(* Logix 5000 project; controller PBS_Perfusion vendor 1 type 14 code 217 rev 32.14; software revision 32.03; part 20 of 27 *)
(* tags used below, declared in another part *)
   Inp_PermOK : BOOL;   // 1=Permissives OK, Valve can energize
   Inp_NBPermOK : BOOL;   // 1=Non-Bypassable Permissives OK, valve can energize
   Inp_IOFault : BOOL;   // Input Communication Status 0=OK, 1=fail
   Inp_Sim : BOOL;   // 1=Simulate working valve; 0=Open/Close/ Monitor actual valve
   Inp_OvrdCmd : DINT;   // Override Mode Command: 0=None, 1=Close, 2=Open
   Cfg_FailOpen : BOOL;   // 1=Fail Open (energize to close), 0=Fail Closed (energize to open)
   Cfg_HasOpenLS : BOOL;   // 1=Valve provides an Open Limit Switch signal
   Cfg_HasClosedLS : BOOL;   // 1=Valve provides a Closed Limit Switch signal
   Cfg_UseOpenLS : BOOL;   // 1=Valve Open LS should be used for failure checking
   Cfg_UseClosedLS : BOOL;   // 1=Valve Closed LS should be used for failure checking
   Cfg_OCmdResets : BOOL;   // 1=New valve OCmd resets shed latches and cleared alarms, 0=OCmdReset req'd.
   PSet_Owner : DINT;   // Program Owner Request ID (non-zero) or Release (zero)
   PCmd_Open : BOOL;   // Program Command to Open Valve
   PCmd_Close : BOOL;   // Program Command to Close Valve
   PCmd_Reset : BOOL;   // Program Command to ResetShed Latches and Cleared Alarms
   XCmd_Open : BOOL;   // External Command to Open Valve
   XCmd_Close : BOOL;   // External Command to Close Valve
   XCmd_Reset : BOOL;   // Ext Cmd to clear shed latches and cleared alarms
   Out : BOOL;   // 1=Energize Valve Solenoid
   Out_Horn : BOOL;   // 1=Sound audible prior to commanded motor start
   SrcQ_IO : DINT;   // Source and Quality of primary I/O (enumeration)
   SrcQ : DINT;   // Source and Quality of primary Val/Sts (enumeration)
   Val_Cmd : DINT;   // Device Command 0=None, 1=Close, 2=Open
   Val_Fdbk : DINT;   // Device Feedback 0=Moving, 1=Closed, 2=Opened, 3=Limit Switch Failure
   Val_Sts : DINT;   // Device Confirmed Sts 0=? 1=Closed 2=Open 5=Closing, 6=Opening
   Val_Fault : DINT;   // Device Fault Status 0=None, 16=Transit Stall, 17 = Full Stall, 32=I/O Fault, 34=Config Error
   Val_NotifyAll : DINT;   // Highest Alarm prio and ack status this object + channel (enum)
   Val_UnackAlmC : DINT;   // Count of Unacknowledged Alarms
   Val_Owner : DINT;   // Current Object Owner ID (0=not owned)
   Sts_Closed : BOOL;   // 1=Valve requested to Close and is confirmed Closed
   Sts_Opening : BOOL;   // 1=Valve requested to open and awaiting open feedback
   Sts_Opened : BOOL;   // 1=Valve requested to open and is confirmed Opened
   Sts_Closing : BOOL;   // 1=Valve requested to Close and awaiting Closed feedback
   Sts_Horn : BOOL;   // 1=Valve Horn Active
   Sts_BypActive : BOOL;   // 1=Bypassing Active (Bypassed or Maintenance)
   Sts_NotRdy : BOOL;   // 1=Device Not Ready, see detail bits for reason
   Nrdy_CfgErr : BOOL;   // 1=Device Not Ready: Configuration Error
   Nrdy_Fail : BOOL;   // 1=Device Not Ready: Device Failure (Shed Requires Reset)
   Nrdy_IOFault : BOOL;   // 1=Device Not Ready: I/O Fault (Shed Requires Reset)
   Sts_AlmInh : BOOL;   // 1=An Alarm is Shelved, Disabled or Suppressed, display icon
   Sts_Err : BOOL;   // 1=Error in Config: see detail bits for reason
   Err_Alarm : BOOL;   // 1=Error in Config: Alarm Min On Time, Shelf Time, Severity
   Sts_Hand : ALIAS FOR CmdSrc.Sts_Hand;
   Sts_OoS : ALIAS FOR CmdSrc.Sts_OoS;
   Sts_Maint : ALIAS FOR CmdSrc.Sts_Maint;
   Sts_Oper : ALIAS FOR CmdSrc.Sts_Oper;
   Sts_RdyReset : ALIAS FOR ORdy_Reset;   // 1=A latched alarm or shed condition is ready to be reset
   Sts_RdyAck : BOOL;   // 1=An alarm is ready to be acknowledged
   Sts_FullStall : ALIAS FOR FullStall.Inp;   // 1=Valve Full Stall (failed to move at all)
   Sts_TransitStall : ALIAS FOR TransitStall.Inp;   // 1=Valve Transit Stall (did not reach target position)
   Sts_IOFault : ALIAS FOR IOFault.Inp;   // I/O Comm Fault Status (0=OK, 1=Bad)
   P_ValveSO : BOOL;   // Unique Parameter Name for auto - discovery
   CmdSrc : P_CmdSrc;   // Valve Mode Selection
   IOFault : P_Alarm;   // I/O Fault Alarm
   IntlkTrip : P_Alarm;   // Interlock Trip Alarm
   TransitStall : P_Alarm;   // Valve Transit Stall (moved but did not reach target) Alarm
   FullStall : P_Alarm;   // Valve Full Stall (did not move) Alarm
   Wrk_Open : BOOL;   // 1=Requested to OPEN Valve, 0=Requested to CLOSE Valve
   Wrk_SimOpenT : TIMER;   // Simulation Delay until Opened
   Wrk_SimCloseT : TIMER;   // Simulation Delay until Closed
   Wrk_OpenFdbk : BOOL;   // 1=LS Feedback shows valve confirmed open
   Wrk_Notify : DINT;   // Buffer for building Val_Notify
   Wrk_ClosedFdbk : BOOL;   // 1=LS Feedback shows valve confirmed closed
   Wrk_TransitStallT : TIMER;   // Timer for Transit Stall Check
   Wrk_FullStallT : TIMER;   // Timer for Full Stall Check
   Wrk_Cmd : DINT;   // Buffer for building Val_Cmd
   Wrk_Sts : DINT;   // Buffer for building Val_Sts
   Wrk_Fault : DINT;   // Buffer for building Val_Fault
   Wrk_SimOpenLS : BOOL;   // Simulated valve Open Limit Switch
   Wrk_SimClosedLS : BOOL;   // Simulated valve Closed Limit Switch
   Wrk_SrcQ : DINT;   // Register for building Source / Quality enumeration
   Val_Notify : DINT;   // Current Alarm Level and Acknowledgement (enumeration)
   Wrk_NotRdy : BOOL;   // Device Not Ready conditions excluding shed latches
   Wrk_NoLongerSim : BOOL;   // Switched from Simulated to Real Valve this scan
   OCmd_Close : BOOL;   // Operator Command to Close Valve
   OCmd_Open : BOOL;   // Operator Command to Open Valve
   ORdy_ResetAckAll : BOOL;   // 1=Ready for OCmd_ResetAckAll (enables HMI button)
   ORdy_Reset : BOOL;   // 1=Ready for OCmd_Reset (enables HMI button)
   MRdy_Check : BOOL;   // 1=Ready for MCmd_Check (enables HMI button)
   MRdy_Bypass : BOOL;   // 1=Ready for MCmd_Bypass (enables HMI button)
   ORdy_Close : BOOL;   // 1=Ready for OCmd_Close (enables HMI button)
   ORdy_Open : BOOL;   // 1=Ready for OCmd_Open (enables HMI button)
   MCmd_Check : BOOL;   // Maintenance Command to Check (not bypass) all Interlocks and Permissives
   MCmd_Bypass : BOOL;   // Maintenance Command to Bypass all Bypassable Interlocks and Permissives
   OCmd_ResetAckAll : BOOL;   // Oper Cmd to reset shed latches and cleared alarms, plus Acknowledge alarms
   OCmd_Reset : BOOL;   // Oper Cmd to clear shed latches and cleared alarms
   Wrk_UnackAlmC : DINT;   // Buffer for building Val_UnackAlmC
   Wrk_CloseCmdRcvd : BOOL;   // 1=Received a Close command this scan
   Wrk_OpenCmdRcvd : BOOL;   // 1=Received an Open command this scan
   Wrk_StartHornT : TIMER;   // Timer for audible alert on start
   Wrk_StartHorn : BOOL;   // 1=Sound audible prior to commanded motor start
   ONS : DINT[3];
(* P_ValveSO, continued *)

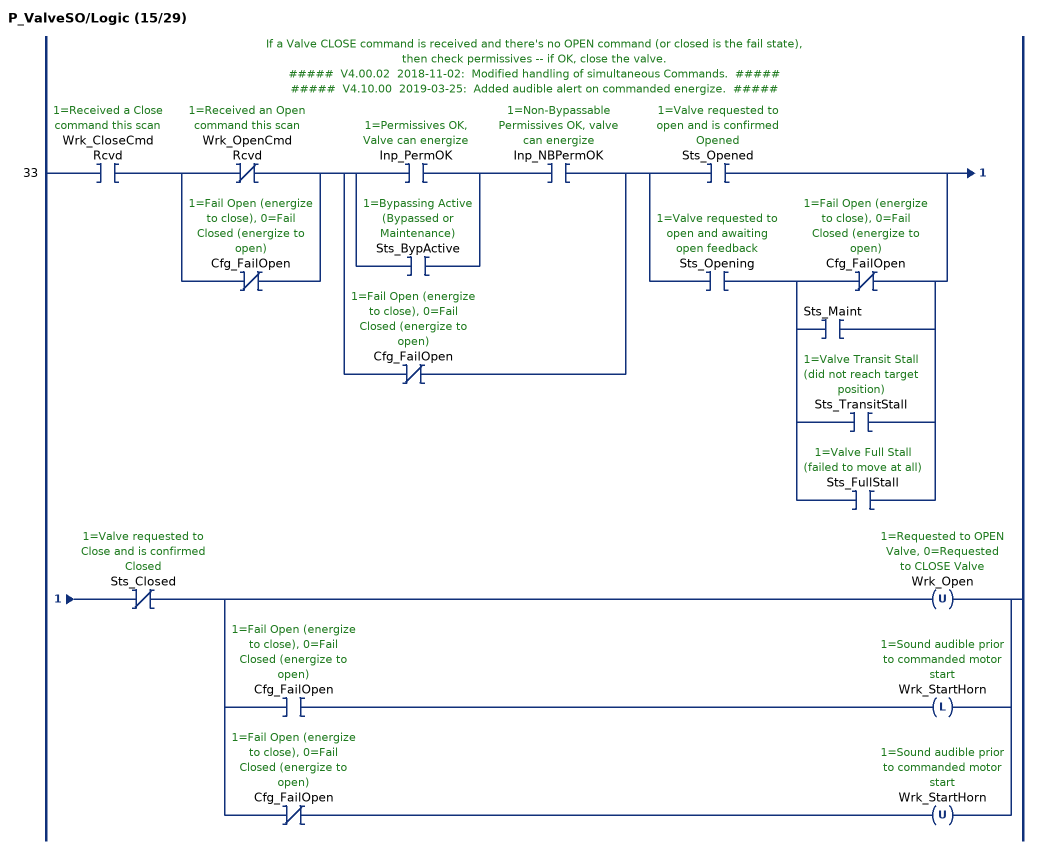
   [picture p443: P_ValveSO/Logic rungs 33-33]
   // If a Valve CLOSE command is received and there's no OPEN command (or closed is the fail state),
   // then check permissives -- if OK, close the valve.
   // #####  V4.00.02  2018-11-02:  Modified handling of simultaneous Commands.  #####
   // #####  V4.10.00  2019-03-25:  Added audible alert on commanded energize.  #####
   33: XIC(Wrk_CloseCmdRcvd)[XIO(Wrk_OpenCmdRcvd) ,XIO(Cfg_FailOpen) ][[XIC(Inp_PermOK) ,XIC(Sts_BypActive) ] XIC(Inp_NBPermOK) ,XIO(Cfg_FailOpen) ][XIC(Sts_Opened) ,XIC(Sts_Opening) [XIO(Cfg_FailOpen) ,XIC(Sts_Maint) ,XIC(Sts_TransitStall) ,XIC(Sts_FullStall) ] ]XIO(Sts_Closed)[OTU(Wrk_Open) ,XIC(Cfg_FailOpen) OTL(Wrk_StartHorn) ,XIO(Cfg_FailOpen) OTU(Wrk_StartHorn) ];
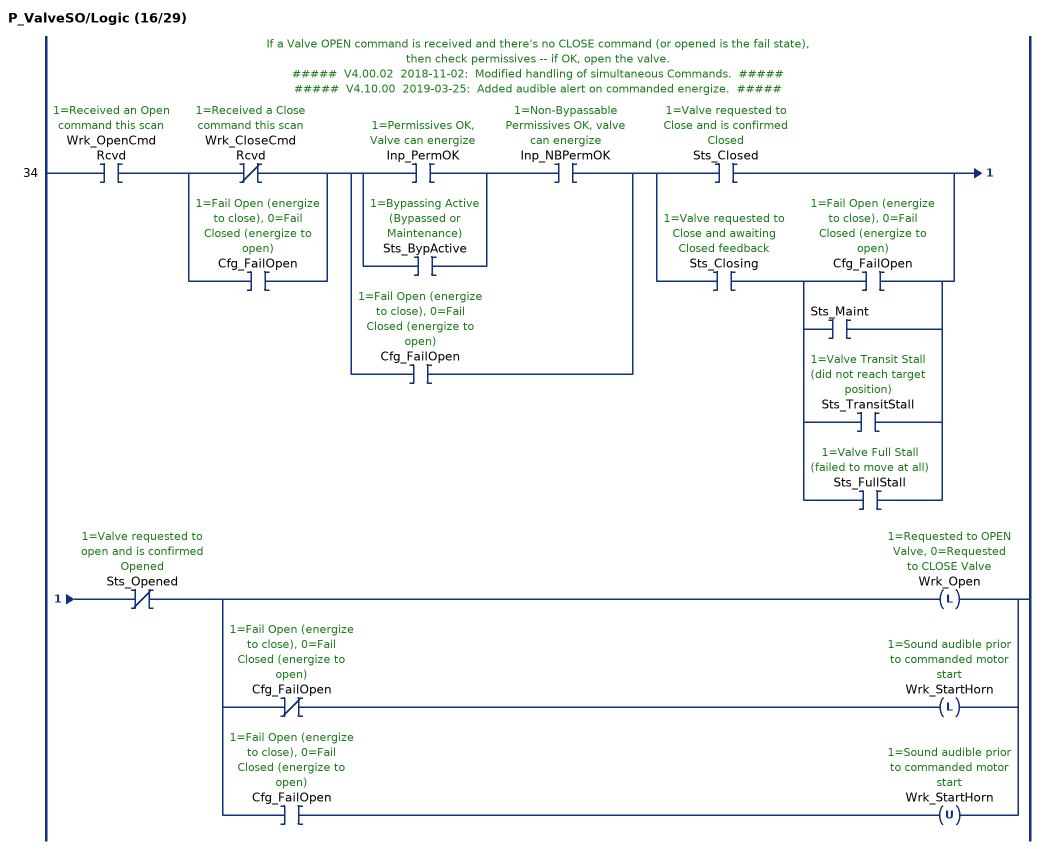
   // If a Valve OPEN command is received and there's no CLOSE command (or opened is the fail state),
   // then check permissives -- if OK, open the valve.
   // #####  V4.00.02  2018-11-02:  Modified handling of simultaneous Commands.  #####
   // #####  V4.10.00  2019-03-25:  Added audible alert on commanded energize.  #####
   34: XIC(Wrk_OpenCmdRcvd)[XIO(Wrk_CloseCmdRcvd) ,XIC(Cfg_FailOpen) ][[XIC(Inp_PermOK) ,XIC(Sts_BypActive) ] XIC(Inp_NBPermOK) ,XIC(Cfg_FailOpen) ][XIC(Sts_Closed) ,XIC(Sts_Closing) [XIC(Cfg_FailOpen) ,XIC(Sts_Maint) ,XIC(Sts_TransitStall) ,XIC(Sts_FullStall) ] ]XIO(Sts_Opened)[OTL(Wrk_Open) ,XIO(Cfg_FailOpen) OTL(Wrk_StartHorn) ,XIC(Cfg_FailOpen) OTU(Wrk_StartHorn) ];
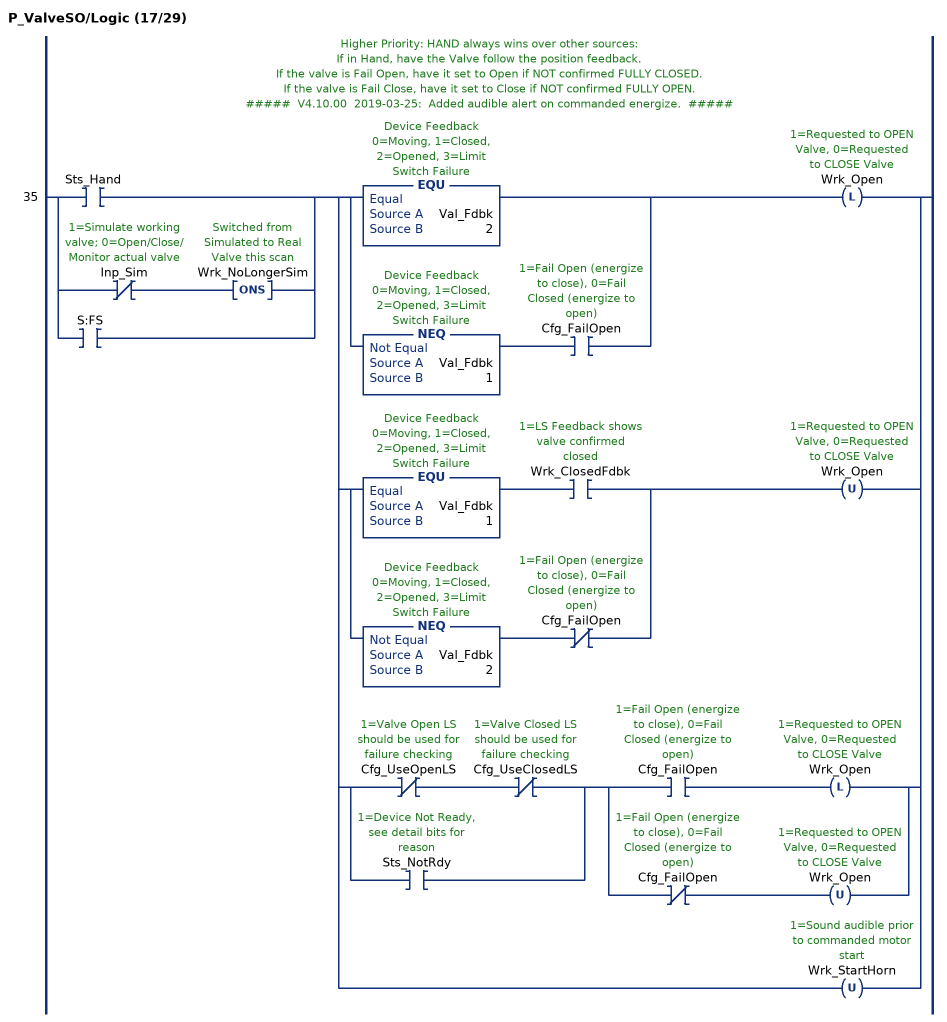
   // Higher Priority: HAND always wins over other sources:
   // If in Hand, have the Valve follow the position feedback.
   // If the valve is Fail Open, have it set to Open if NOT confirmed FULLY CLOSED.
   // If the valve is Fail Close, have it set to Close if NOT confirmed FULLY OPEN.
   // #####  V4.10.00  2019-03-25:  Added audible alert on commanded energize.  #####
   35: [XIC(Sts_Hand) ,XIO(Inp_Sim) ONS(Wrk_NoLongerSim) ,XIC(S:FS) ][[EQU(Val_Fdbk,2) ,NEQ(Val_Fdbk,1) XIC(Cfg_FailOpen) ] OTL(Wrk_Open) ,[EQU(Val_Fdbk,1) XIC(Wrk_ClosedFdbk) ,NEQ(Val_Fdbk,2) XIO(Cfg_FailOpen) ] OTU(Wrk_Open) ,[XIO(Cfg_UseOpenLS) XIO(Cfg_UseClosedLS) ,XIC(Sts_NotRdy) ] [XIC(Cfg_FailOpen) OTL(Wrk_Open) ,XIO(Cfg_FailOpen) OTU(Wrk_Open) ] ,OTU(Wrk_StartHorn) ];
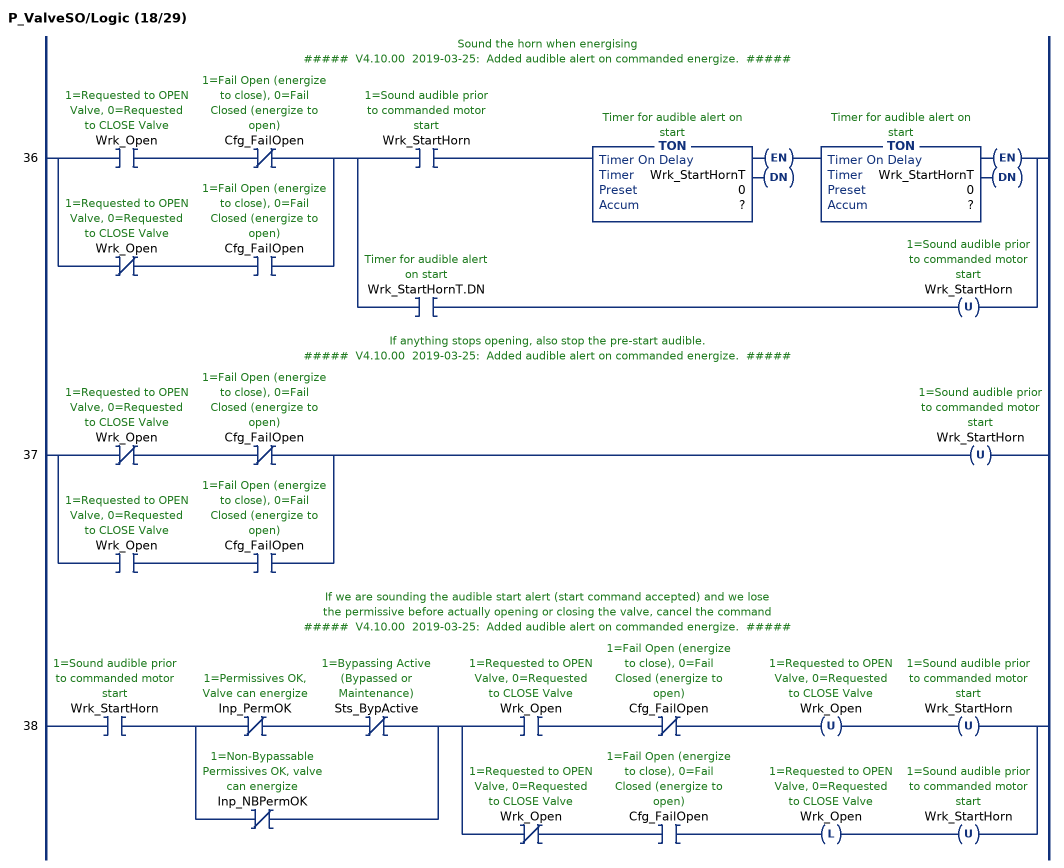
   // Sound the horn when energising
   // #####  V4.10.00  2019-03-25:  Added audible alert on commanded energize.  #####
   36: [XIC(Wrk_Open) XIO(Cfg_FailOpen) ,XIO(Wrk_Open) XIC(Cfg_FailOpen) ][XIC(Wrk_StartHorn) TON(Wrk_StartHornT,?,?) TON(Wrk_StartHornT,?,?) ,XIC(Wrk_StartHornT.DN) OTU(Wrk_StartHorn) ];
   // If anything stops opening, also stop the pre-start audible.
   // #####  V4.10.00  2019-03-25:  Added audible alert on commanded energize.  #####
   37: [XIO(Wrk_Open) XIO(Cfg_FailOpen) ,XIC(Wrk_Open) XIC(Cfg_FailOpen) ]OTU(Wrk_StartHorn);
   // If we are sounding the audible start alert (start command accepted) and we lose
   // the permissive before actually opening or closing the valve, cancel the command
   // #####  V4.10.00  2019-03-25:  Added audible alert on commanded energize.  #####
   38: XIC(Wrk_StartHorn)[XIO(Inp_PermOK) XIO(Sts_BypActive) ,XIO(Inp_NBPermOK) ][XIC(Wrk_Open) XIO(Cfg_FailOpen) OTU(Wrk_Open) OTU(Wrk_StartHorn) ,XIO(Wrk_Open) XIC(Cfg_FailOpen) OTL(Wrk_Open) OTU(Wrk_StartHorn) ];
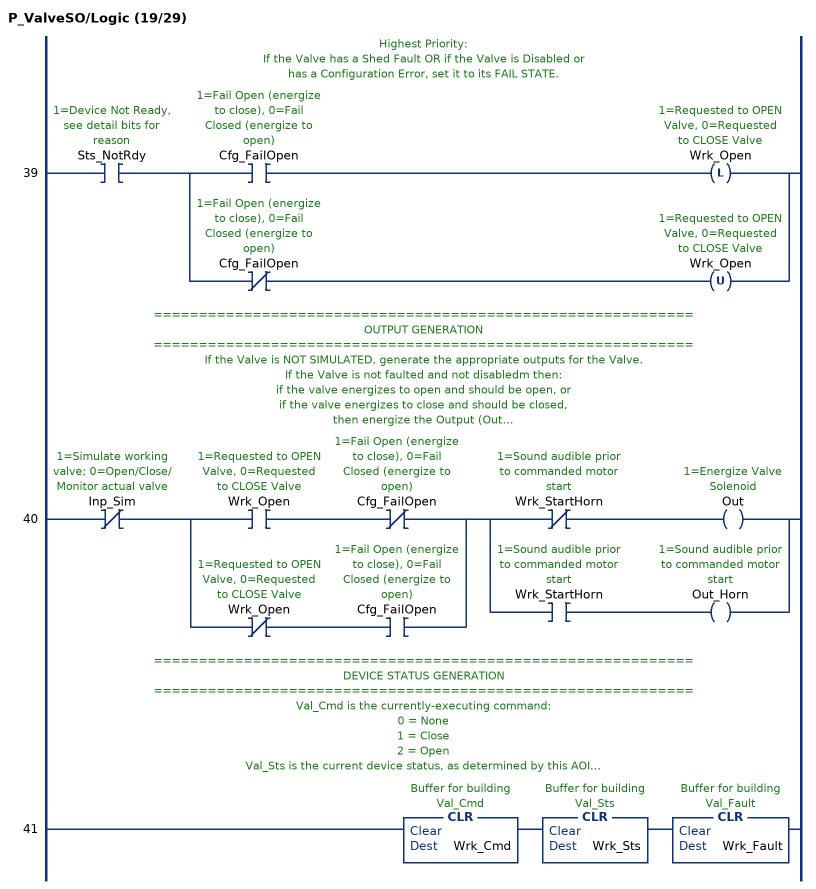
   // Highest Priority:
   // If the Valve has a Shed Fault OR if the Valve is Disabled or
   // has a Configuration Error, set it to its FAIL STATE.
   39: XIC(Sts_NotRdy)[XIC(Cfg_FailOpen) OTL(Wrk_Open) ,XIO(Cfg_FailOpen) OTU(Wrk_Open) ];
   // ============================================================
   // OUTPUT GENERATION
   // ============================================================
   // If the Valve is NOT SIMULATED, generate the appropriate outputs for the Valve.
   // If the Valve is not faulted and not disabledm then:
   // if the valve energizes to open and should be open, or
   // if the valve energizes to close and should be closed,
   // then energize the Output (Out)
   // #####  V4.10.00  2019-03-25:  Added audible alert on commanded energize.  #####
   40: XIO(Inp_Sim)[XIC(Wrk_Open) XIO(Cfg_FailOpen) ,XIO(Wrk_Open) XIC(Cfg_FailOpen) ][XIO(Wrk_StartHorn) OTE(Out) ,XIC(Wrk_StartHorn) OTE(Out_Horn) ];
   // ============================================================
   // DEVICE STATUS GENERATION
   // ============================================================
   // Val_Cmd is the currently-executing command:
   // 0 = None
   // 1 = Close
   // 2 = Open
   // Val_Sts is the current device status, as determined by this AOI,
   // based on its knowledge of commands executed and feedback.
   // (This is the status that should be monitored by, for example, FT Historian.)
   // 0 = Powerup / Unknown
   // 1 = Closed
   // 2 = Opened
   // 5 = Closing
   // 6 = Opening
   // 10 = Horn
   // 33 = Out of Service
   // Val_Fault is the current device fault status, as determined by this AOI,
   // based on its knowledge of commands executed and feedback.
   // (This is the fault status that should be monitored by, for example, FT Historian.)
   // 0 = None
   // 16 = Full Stall
   // 17 = Transit Stall
   // 32 = I/O Fault (from Input)
   // 34 = Configuration Error
   // #####  V4.10.00  2019-03-25:  Added Horn Status.  #####
   41: CLR(Wrk_Cmd)CLR(Wrk_Sts)CLR(Wrk_Fault);
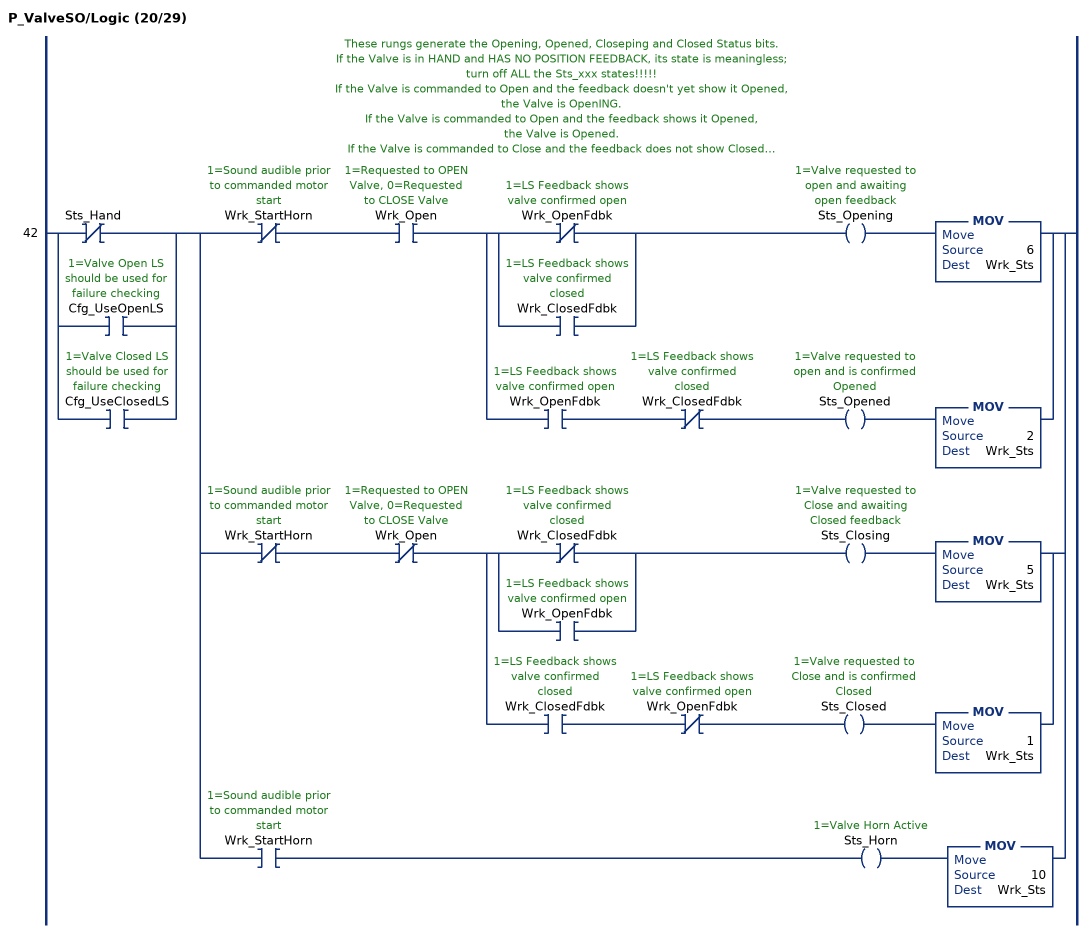
   // These rungs generate the Opening, Opened, Closeping and Closed Status bits.
   // If the Valve is in HAND and HAS NO POSITION FEEDBACK, its state is meaningless;
   // turn off ALL the Sts_xxx states!!!!!
   // If the Valve is commanded to Open and the feedback doesn't yet show it Opened,
   // the Valve is OpenING.
   // If the Valve is commanded to Open and the feedback shows it Opened,
   // the Valve is Opened.
   // If the Valve is commanded to Close and the feedback does not show Closed,
   // the Valve is CloseING.
   // If the Valve is commanded to Close and the feedback shows it has Closed,
   // the Valve is Closed.
   // If the audible alert is active, show the Status as HORN.
   // #####  V4.10.00  2019-03-25:  Added Horn Status.  #####
   42: [XIO(Sts_Hand) ,XIC(Cfg_UseOpenLS) ,XIC(Cfg_UseClosedLS) ][XIO(Wrk_StartHorn) XIC(Wrk_Open) [[XIO(Wrk_OpenFdbk) ,XIC(Wrk_ClosedFdbk) ] OTE(Sts_Opening) MOV(6,Wrk_Sts) ,XIC(Wrk_OpenFdbk) XIO(Wrk_ClosedFdbk) OTE(Sts_Opened) MOV(2,Wrk_Sts) ] ,XIO(Wrk_StartHorn) XIO(Wrk_Open) [[XIO(Wrk_ClosedFdbk) ,XIC(Wrk_OpenFdbk) ] OTE(Sts_Closing) MOV(5,Wrk_Sts) ,XIC(Wrk_ClosedFdbk) XIO(Wrk_OpenFdbk) OTE(Sts_Closed) MOV(1,Wrk_Sts) ] ,XIC(Wrk_StartHorn) OTE(Sts_Horn) MOV(10,Wrk_Sts) ];
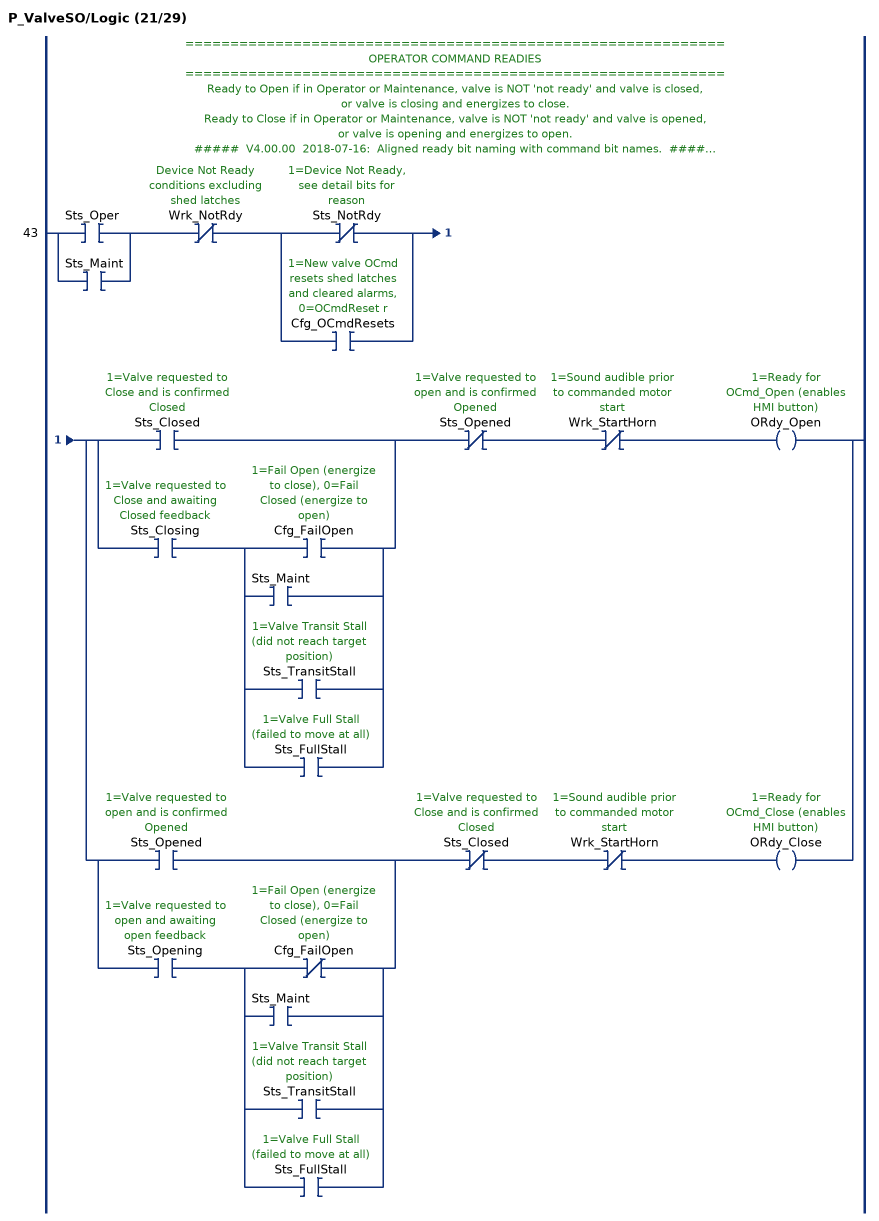
   // ============================================================
   // OPERATOR COMMAND READIES
   // ============================================================
   // Ready to Open if in Operator or Maintenance, valve is NOT 'not ready' and valve is closed,
   // or valve is closing and energizes to close.
   // Ready to Close if in Operator or Maintenance, valve is NOT 'not ready' and valve is opened,
   // or valve is opening and energizes to open.
   // #####  V4.00.00  2018-07-16:  Aligned ready bit naming with command bit names.  #####
   // #####  V4.10.00  2019-03-25:  Added audible alert on commanded energize.  #####
   43: [XIC(Sts_Oper) ,XIC(Sts_Maint) ]XIO(Wrk_NotRdy)[XIO(Sts_NotRdy) ,XIC(Cfg_OCmdResets) ][[XIC(Sts_Closed) ,XIC(Sts_Closing) [XIC(Cfg_FailOpen) ,XIC(Sts_Maint) ,XIC(Sts_TransitStall) ,XIC(Sts_FullStall) ] ] XIO(Sts_Opened) XIO(Wrk_StartHorn) OTE(ORdy_Open) ,[XIC(Sts_Opened) ,XIC(Sts_Opening) [XIO(Cfg_FailOpen) ,XIC(Sts_Maint) ,XIC(Sts_TransitStall) ,XIC(Sts_FullStall) ] ] XIO(Sts_Closed) XIO(Wrk_StartHorn) OTE(ORdy_Close) ];
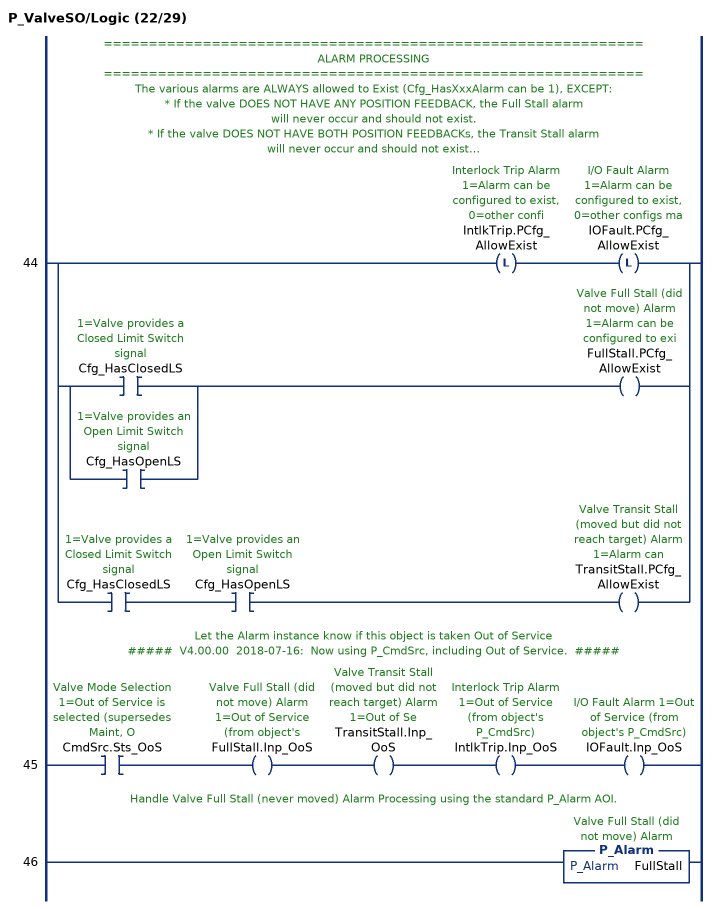
   // ============================================================
   // ALARM PROCESSING
   // ============================================================
   // The various alarms are ALWAYS allowed to Exist (Cfg_HasXxxAlarm can be 1), EXCEPT:
   // * If the valve DOES NOT HAVE ANY POSITION FEEDBACK, the Full Stall alarm
   // will never occur and should not exist.
   // * If the valve DOES NOT HAVE BOTH POSITION FEEDBACKs, the Transit Stall alarm
   // will never occur and should not exist.
   // (If feedback exists, the stall alarms must be allowed to exist.)
   // #####  V4.00.00  2018-07-16:  Deleted Cfg_PCmdClear; all Program Commands are now self-clearing.  #####
   44: [OTL(IntlkTrip.PCfg_AllowExist) OTL(IOFault.PCfg_AllowExist) ,[XIC(Cfg_HasClosedLS) ,XIC(Cfg_HasOpenLS) ] OTE(FullStall.PCfg_AllowExist) ,XIC(Cfg_HasClosedLS) XIC(Cfg_HasOpenLS) OTE(TransitStall.PCfg_AllowExist) ];
   // Let the Alarm instance know if this object is taken Out of Service
   // #####  V4.00.00  2018-07-16:  Now using P_CmdSrc, including Out of Service.  #####
   45: XIC(CmdSrc.Sts_OoS)OTE(FullStall.Inp_OoS)OTE(TransitStall.Inp_OoS)OTE(IntlkTrip.Inp_OoS)OTE(IOFault.Inp_OoS);
   // Handle Valve Full Stall (never moved) Alarm Processing using the standard P_Alarm AOI.
   46: P_Alarm(FullStall);
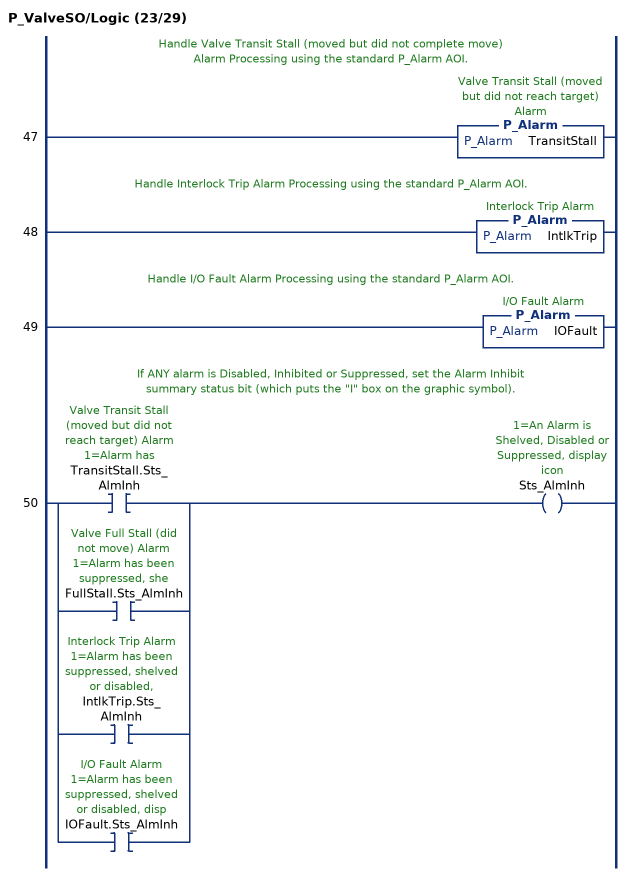
   // Handle Valve Transit Stall (moved but did not complete move)
   // Alarm Processing using the standard P_Alarm AOI.
   47: P_Alarm(TransitStall);
   // Handle Interlock Trip Alarm Processing using the standard P_Alarm AOI.
   48: P_Alarm(IntlkTrip);
   // Handle I/O Fault Alarm Processing using the standard P_Alarm AOI.
   49: P_Alarm(IOFault);
   // If ANY alarm is Disabled, Inhibited or Suppressed, set the Alarm Inhibit
   // summary status bit (which puts the "I" box on the graphic symbol).
   50: [XIC(TransitStall.Sts_AlmInh) ,XIC(FullStall.Sts_AlmInh) ,XIC(IntlkTrip.Sts_AlmInh) ,XIC(IOFault.Sts_AlmInh) ]OTE(Sts_AlmInh);
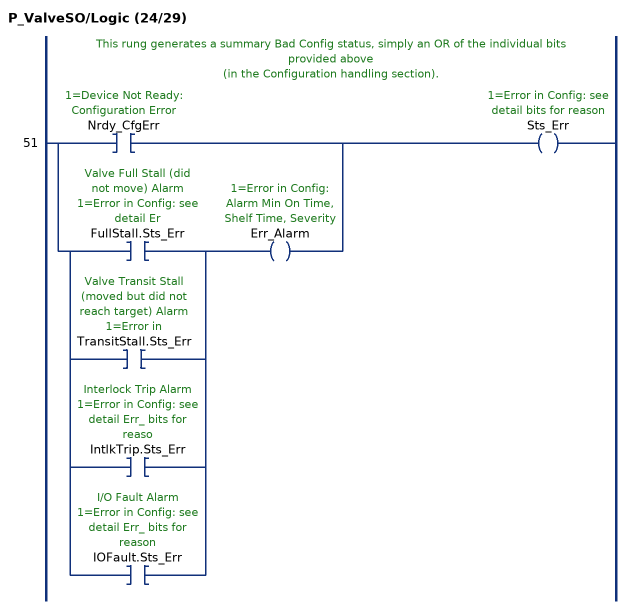
   // This rung generates a summary Bad Config status, simply an OR of the individual bits provided above
   // (in the Configuration handling section).
   51: [XIC(Nrdy_CfgErr) ,[XIC(FullStall.Sts_Err) ,XIC(TransitStall.Sts_Err) ,XIC(IntlkTrip.Sts_Err) ,XIC(IOFault.Sts_Err) ] OTE(Err_Alarm) ]OTE(Sts_Err);
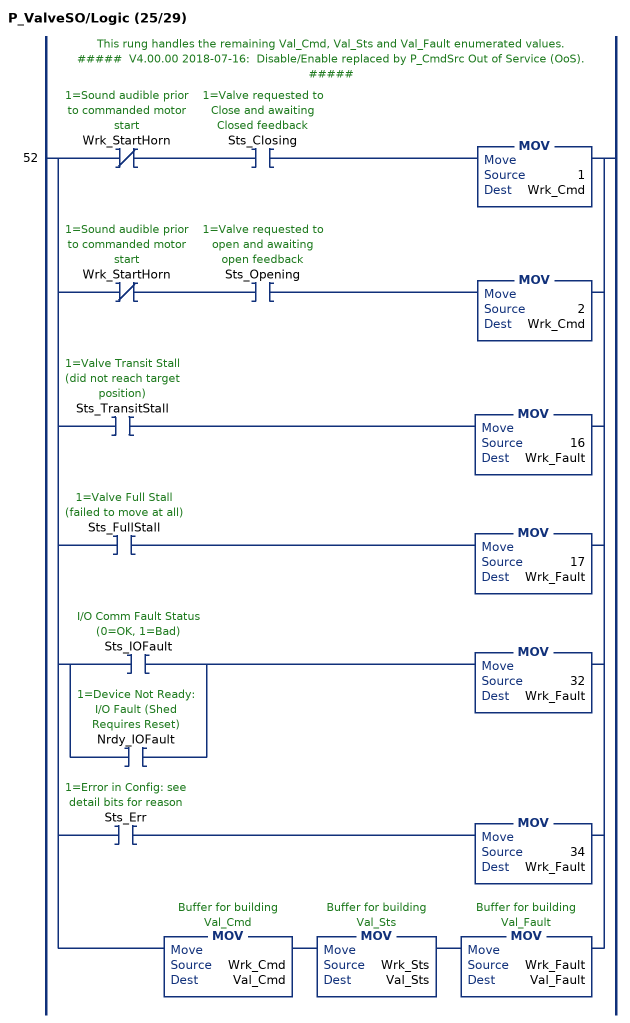
   // This rung handles the remaining Val_Cmd, Val_Sts and Val_Fault enumerated values.
   // #####  V4.00.00 2018-07-16:  Disable/Enable replaced by P_CmdSrc Out of Service (OoS).  #####
   52: [XIO(Wrk_StartHorn) XIC(Sts_Closing) MOV(1,Wrk_Cmd) ,XIO(Wrk_StartHorn) XIC(Sts_Opening) MOV(2,Wrk_Cmd) ,XIC(Sts_TransitStall) MOV(16,Wrk_Fault) ,XIC(Sts_FullStall) MOV(17,Wrk_Fault) ,[XIC(Sts_IOFault) ,XIC(Nrdy_IOFault) ] MOV(32,Wrk_Fault) ,XIC(Sts_Err) MOV(34,Wrk_Fault) ,MOV(Wrk_Cmd,Val_Cmd) MOV(Wrk_Sts,Val_Sts) MOV(Wrk_Fault,Val_Fault) ];
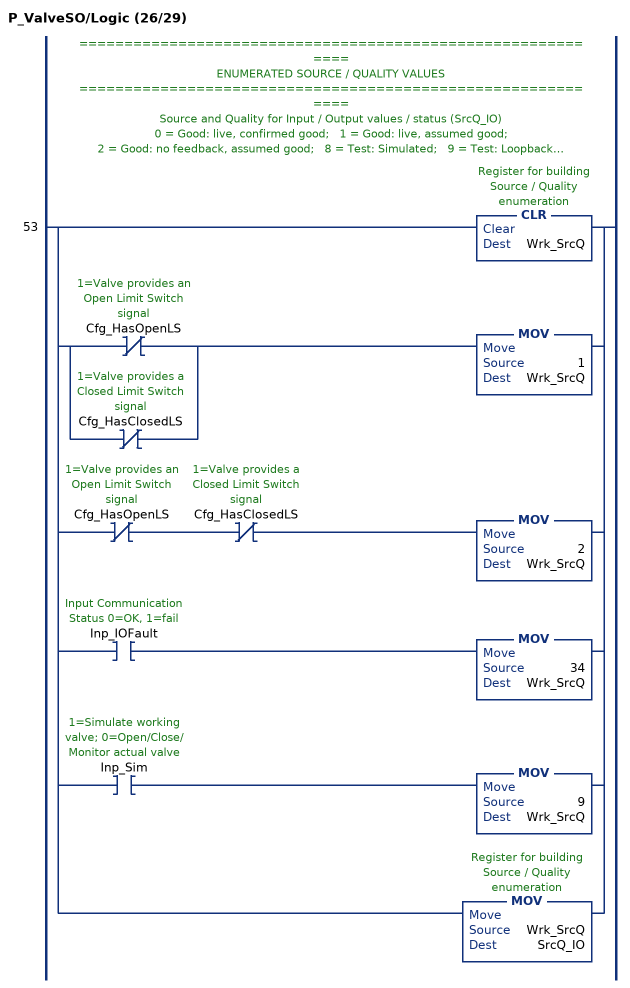
   // ============================================================
   // ENUMERATED SOURCE / QUALITY VALUES
   // ============================================================
   // Source and Quality for Input / Output values / status (SrcQ_IO)
   // 0 = Good: live, confirmed good;   1 = Good: live, assumed good;
   // 2 = Good: no feedback, assumed good;   8 = Test: Simulated;   9 = Test: Loopback;
   // 10 = Test: Manually Entered;   16 = Uncertain: Live, off-spec;
   // 17 = Uncertain, Substituted at Device / Bus;   18 = Uncertain, Substituted at AOI;
   // 19 = Uncertain, using last known good;    20 = Uncertain, using replacement value;
   // 32 = Bad, Signal Failure;   33 = Bad, Channel Fault;
   // 34 = Bad, Module / Comms Fault;   35 = Bad, Invalid Configuration
   53: [CLR(Wrk_SrcQ) ,[XIO(Cfg_HasOpenLS) ,XIO(Cfg_HasClosedLS) ] MOV(1,Wrk_SrcQ) ,XIO(Cfg_HasOpenLS) XIO(Cfg_HasClosedLS) MOV(2,Wrk_SrcQ) ,XIC(Inp_IOFault) MOV(34,Wrk_SrcQ) ,XIC(Inp_Sim) MOV(9,Wrk_SrcQ) ,MOV(Wrk_SrcQ,SrcQ_IO) ];
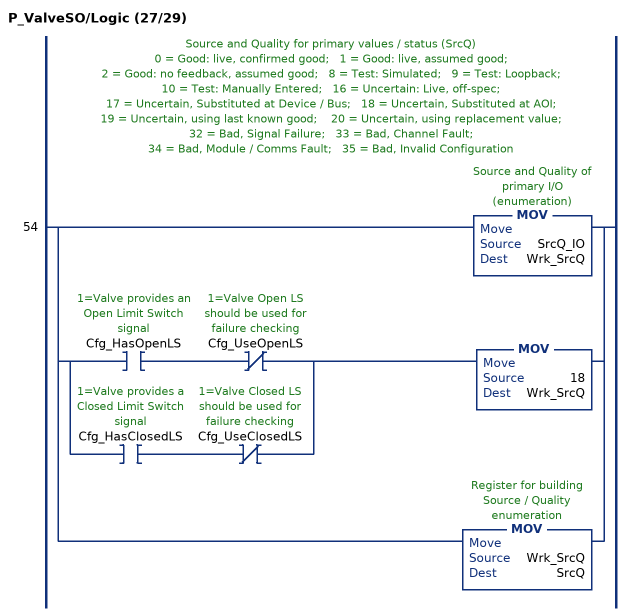
   // Source and Quality for primary values / status (SrcQ)
   // 0 = Good: live, confirmed good;   1 = Good: live, assumed good;
   // 2 = Good: no feedback, assumed good;   8 = Test: Simulated;   9 = Test: Loopback;
   // 10 = Test: Manually Entered;   16 = Uncertain: Live, off-spec;
   // 17 = Uncertain, Substituted at Device / Bus;   18 = Uncertain, Substituted at AOI;
   // 19 = Uncertain, using last known good;    20 = Uncertain, using replacement value;
   // 32 = Bad, Signal Failure;   33 = Bad, Channel Fault;
   // 34 = Bad, Module / Comms Fault;   35 = Bad, Invalid Configuration
   54: [MOV(SrcQ_IO,Wrk_SrcQ) ,[XIC(Cfg_HasOpenLS) XIO(Cfg_UseOpenLS) ,XIC(Cfg_HasClosedLS) XIO(Cfg_UseClosedLS) ] MOV(18,Wrk_SrcQ) ,MOV(Wrk_SrcQ,SrcQ) ];
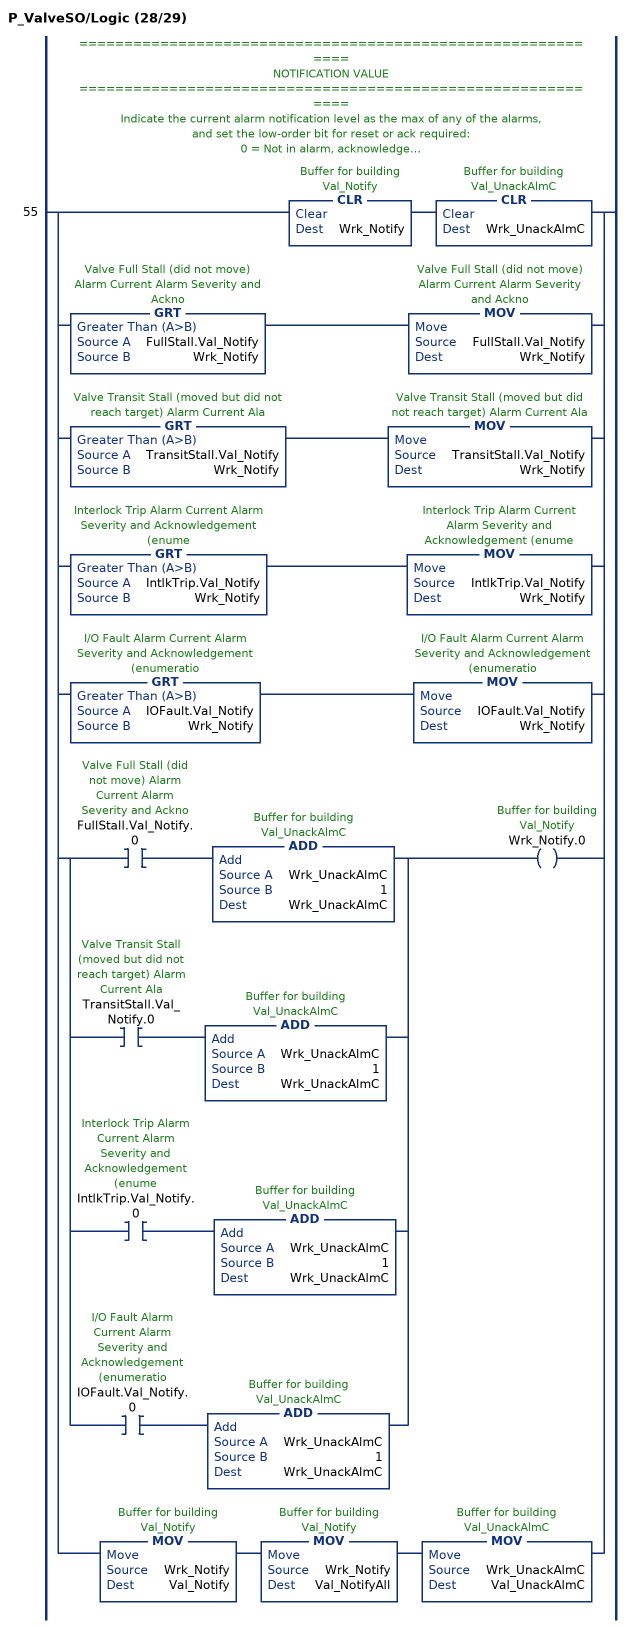
   // ============================================================
   // NOTIFICATION VALUE
   // ============================================================
   // Indicate the current alarm notification level as the max of any of the alarms,
   // and set the low-order bit for reset or ack required:
   // 0 = Not in alarm, acknowledged
   // 1 = Not in alarm, unacknowledged or reset required
   // 2 = Low severity alarm, acknowledged
   // 3 = Low severity alarm, unacknowledged
   // 4 = Medium severity alarm, acknowledged
   // 5 = Medium severity alarm, unacknowledged
   // 6 = High severity alarm, acknowledged
   // 7 = High severity alarm, unacknowledged
   // 8 = Urgent severity alarm, acknowledged
   // 9 = Urgent severity alarm, unacknowledged
   // #####  V4.00.00  2018-07-16:  Added Val_NotifyAll and Val_UnackAlmC to roll up alarm  #####
   // #####  priority / ack status and unack. alarm count.  #####
   55: [CLR(Wrk_Notify) CLR(Wrk_UnackAlmC) ,GRT(FullStall.Val_Notify,Wrk_Notify) MOV(FullStall.Val_Notify,Wrk_Notify) ,GRT(TransitStall.Val_Notify,Wrk_Notify) MOV(TransitStall.Val_Notify,Wrk_Notify) ,GRT(IntlkTrip.Val_Notify,Wrk_Notify) MOV(IntlkTrip.Val_Notify,Wrk_Notify) ,GRT(IOFault.Val_Notify,Wrk_Notify) MOV(IOFault.Val_Notify,Wrk_Notify) ,[XIC(FullStall.Val_Notify.0) ADD(Wrk_UnackAlmC,1,Wrk_UnackAlmC) ,XIC(TransitStall.Val_Notify.0) ADD(Wrk_UnackAlmC,1,Wrk_UnackAlmC) ,XIC(IntlkTrip.Val_Notify.0) ADD(Wrk_UnackAlmC,1,Wrk_UnackAlmC) ,XIC(IOFault.Val_Notify.0) ADD(Wrk_UnackAlmC,1,Wrk_UnackAlmC) ] OTE(Wrk_Notify.0) ,MOV(Wrk_Notify,Val_Notify) MOV(Wrk_Notify,Val_NotifyAll) MOV(Wrk_UnackAlmC,Val_UnackAlmC) ];
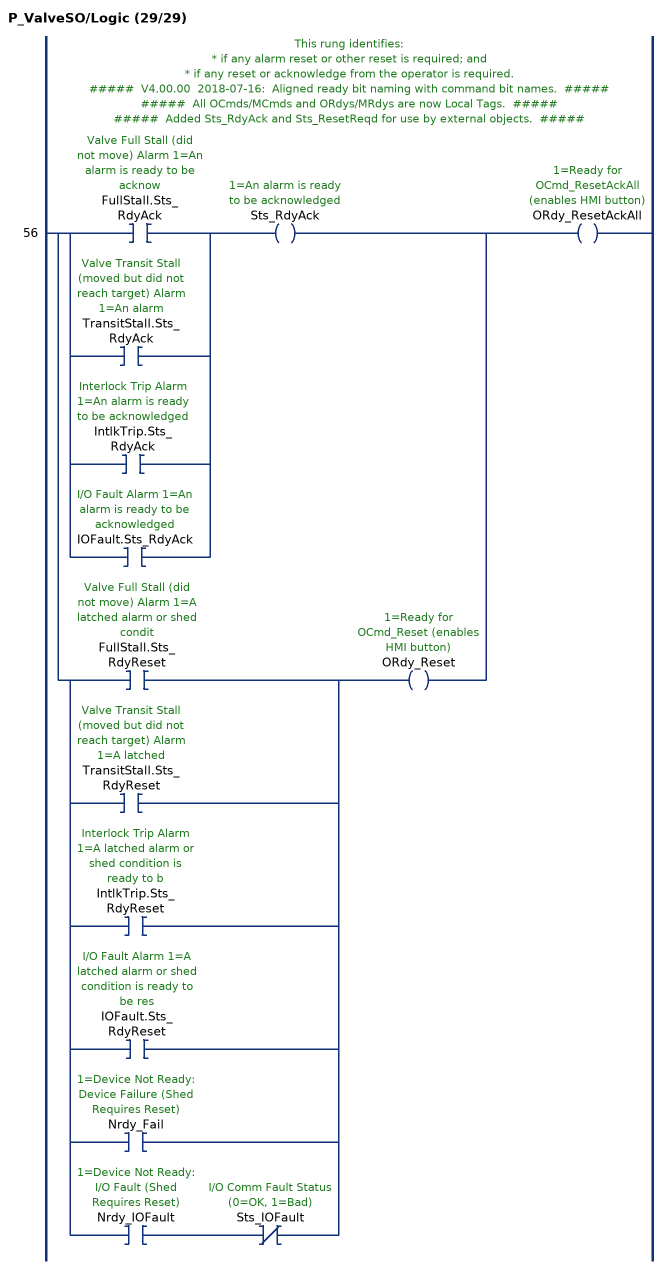
   // This rung identifies:
   // * if any alarm reset or other reset is required; and
   // * if any reset or acknowledge from the operator is required.
   // #####  V4.00.00  2018-07-16:  Aligned ready bit naming with command bit names.  #####
   // #####  All OCmds/MCmds and ORdys/MRdys are now Local Tags.  #####
   // #####  Added Sts_RdyAck and Sts_ResetReqd for use by external objects.  #####
   56: [[XIC(FullStall.Sts_RdyAck) ,XIC(TransitStall.Sts_RdyAck) ,XIC(IntlkTrip.Sts_RdyAck) ,XIC(IOFault.Sts_RdyAck) ] OTE(Sts_RdyAck) ,[XIC(FullStall.Sts_RdyReset) ,XIC(TransitStall.Sts_RdyReset) ,XIC(IntlkTrip.Sts_RdyReset) ,XIC(IOFault.Sts_RdyReset) ,XIC(Nrdy_Fail) ,XIC(Nrdy_IOFault) XIO(Sts_IOFault) ] OTE(ORdy_Reset) ]OTE(ORdy_ResetAckAll);
END_ROUTINE

ROUTINE Prescan   (* ladder *)
// Clear Ownership, set to De-Energized state, clear "lurking" Commands
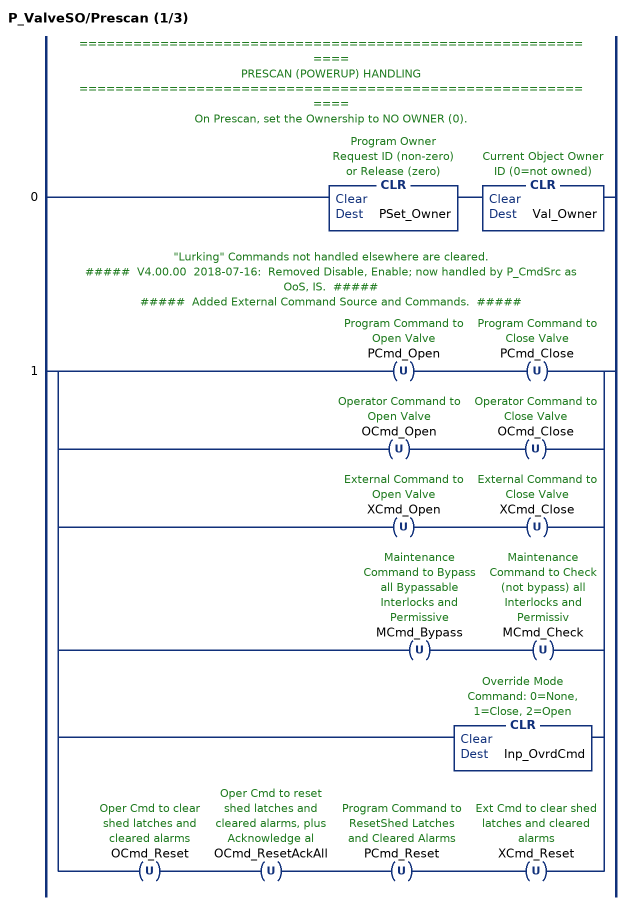
   // ============================================================
   // PRESCAN (POWERUP) HANDLING
   // ============================================================
   // On Prescan, set the Ownership to NO OWNER (0).
   0: CLR(PSet_Owner)CLR(Val_Owner);
   // "Lurking" Commands not handled elsewhere are cleared.
   // #####  V4.00.00  2018-07-16:  Removed Disable, Enable; now handled by P_CmdSrc as OoS, IS.  #####
   // #####  Added External Command Source and Commands.  #####
   1: [OTU(PCmd_Open) OTU(PCmd_Close) ,OTU(OCmd_Open) OTU(OCmd_Close) ,OTU(XCmd_Open) OTU(XCmd_Close) ,OTU(MCmd_Bypass) OTU(MCmd_Check) ,CLR(Inp_OvrdCmd) ,OTU(OCmd_Reset) OTU(OCmd_ResetAckAll) OTU(PCmd_Reset) OTU(XCmd_Reset) ];
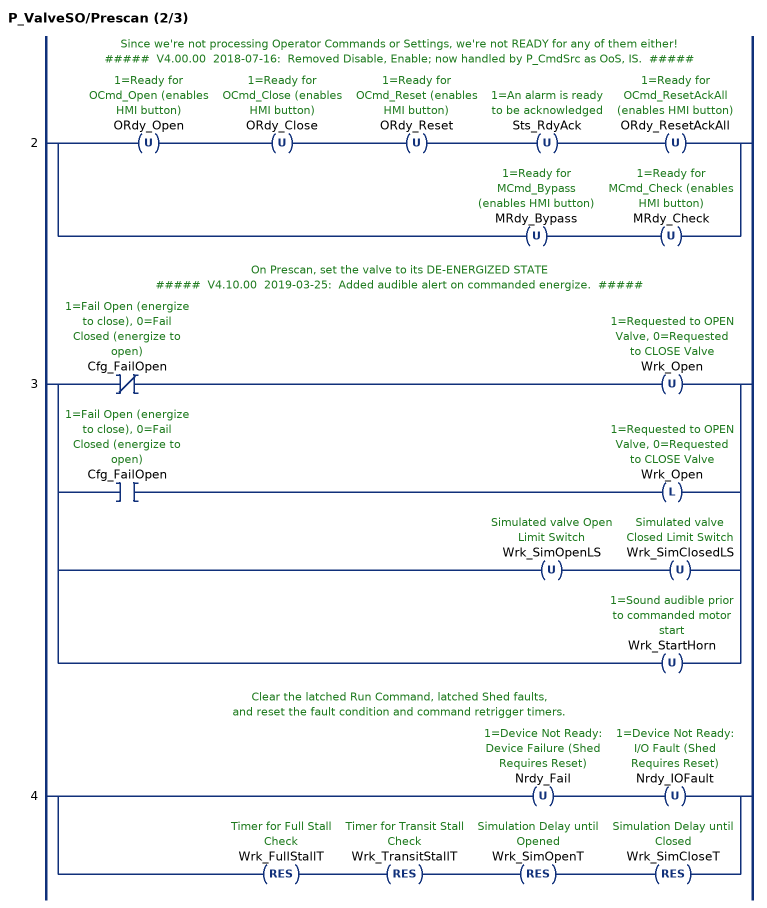
   // Since we're not processing Operator Commands or Settings, we're not READY for any of them either!
   // #####  V4.00.00  2018-07-16:  Removed Disable, Enable; now handled by P_CmdSrc as OoS, IS.  #####
   2: [OTU(ORdy_Open) OTU(ORdy_Close) OTU(ORdy_Reset) OTU(Sts_RdyAck) OTU(ORdy_ResetAckAll) ,OTU(MRdy_Bypass) OTU(MRdy_Check) ];
   // On Prescan, set the valve to its DE-ENERGIZED STATE
   // #####  V4.10.00  2019-03-25:  Added audible alert on commanded energize.  #####
   3: [XIO(Cfg_FailOpen) OTU(Wrk_Open) ,XIC(Cfg_FailOpen) OTL(Wrk_Open) ,OTU(Wrk_SimOpenLS) OTU(Wrk_SimClosedLS) ,OTU(Wrk_StartHorn) ];
   // Clear the latched Run Command, latched Shed faults,
   // and reset the fault condition and command retrigger timers.
   4: [OTU(Nrdy_Fail) OTU(Nrdy_IOFault) ,RES(Wrk_FullStallT) RES(Wrk_TransitStallT) RES(Wrk_SimOpenT) RES(Wrk_SimCloseT) ];
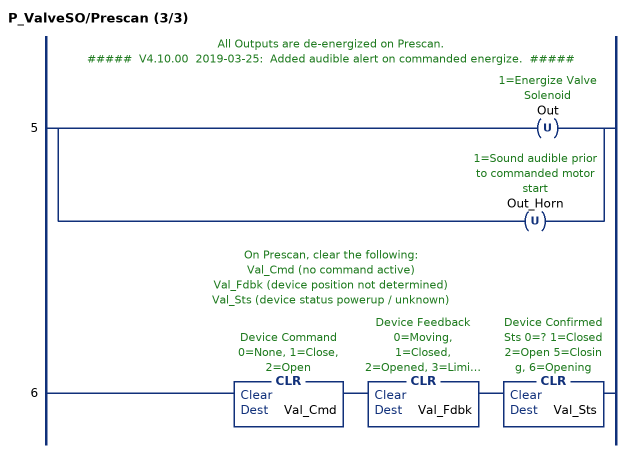
   // All Outputs are de-energized on Prescan.
   // #####  V4.10.00  2019-03-25:  Added audible alert on commanded energize.  #####
   5: [OTU(Out) ,OTU(Out_Horn) ];
   // On Prescan, clear the following:
   // Val_Cmd (no command active)
   // Val_Fdbk (device position not determined)
   // Val_Sts (device status powerup / unknown)
   6: CLR(Val_Cmd)CLR(Val_Fdbk)CLR(Val_Sts);
END_ROUTINE
END_ADD_ON_INSTRUCTION
